// TIA Portal V16 export
// export: Created 2021-09-08T12:46:09.589751Z, ExportSetting WithDefaults, DisplayName Totally Integrated Automation Portal, DisplayVersion V16 Update 3, DisplayName TIA Portal Version Control Interface, DisplayVersion V16 Update 2, DisplayName TIA Portal Openness, DisplayVersion V16 Update 3, DisplayName TIA Portal Teamcenter Gateway, DisplayVersion V16, DisplayName STEP 7 Professional, DisplayVersion V16 Update 3, DisplayName STEP 7 Safety, DisplayVersion V16, DisplayName WinCC Advanced, DisplayVersion V16 Update 3
DATA_BLOCK "dtAnalogData"   // DB1
{ S7_Optimized_Access := 'FALSE' }
VERSION : 0.1
// stored: AutoNumber true, DBAccessibleFromOPCUA true, IsOnlyStoredInLoadMemory false, IsWriteProtectedInAS false
   VAR
      plc_data : Array[0.."PLC_AI"] of "Ai";
      et_data : Array[0.."ET_AI"] of "Ai";
   END_VAR
BEGIN
   // et_data[0] : aiLT201
   // et_data[1] : aiLT202
   // et_data[2] : aiPT301
   // et_data[3] : aiPT401
   // et_data[4] : aiPT501
   // et_data[5] : aiPT502
   // et_data[6] : aiPT503
   // et_data[7] : aiPT504
   // et_data[8] : aiPT505
   // et_data[9] : aiPT506
   // et_data[10] : aiPT507
   // et_data[11] : aiLT601
   // et_data[12] : aiPT701
   // et_data[13] : aiPT901
   // et_data[14] : aiPT902
   // et_data[15] : aiLT1101
   // et_data[16] : aiPT1201
   // et_data[17] : aiPT1301
   // et_data[18] : aiPT1302
   // et_data[19] : aiLT1401
   // et_data[20] : aiLT1402
   // et_data[21] : aiPT1501
   // et_data[22] : aiPT1701
   // et_data[23] : aiLT1801
   // et_data[24] : aiFM501
   // et_data[25] : aiFM502
   // et_data[26] : aiFM901
   // et_data[27] : aiFM902
   // et_data[28] : aiFM1301
   // et_data[29] : aiFM1302
   // et_data[30] : aiORP801
   // et_data[31] : aiCDI901
   // et_data[32] : aiCDI1301
   // et_data[33] : aiCDI1302
   // et_data[34] : aiCDI1801
END_DATA_BLOCK
